(* IEC 61131-3 sources: -3/Library, 1 file *)

(* ---- Library.fun ---- *)
FUNCTION_BLOCK FB_Motor (*TODO: Add your comment here*) (*$GROUP=User,$CAT=User,$GROUPICON=User.png,$CATICON=User.png*)
	VAR_INPUT
		in : REAL;
	END_VAR
	VAR_OUTPUT
		out_w : REAL;
		out_phi : REAL;
	END_VAR
	VAR
		k_e : REAL;
		T_m : REAL;
		dt : REAL;
		integrator : FB_Integrator;
		integrator_phi : FB_Integrator;
	END_VAR
END_FUNCTION_BLOCK

FUNCTION_BLOCK FB_Integrator (*TODO: Add your comment here*) (*$GROUP=User,$CAT=User,$GROUPICON=User.png,$CATICON=User.png*)
	VAR_INPUT
		in : REAL;
		dt : REAL;
	END_VAR
	VAR_OUTPUT
		out : REAL;
	END_VAR
	VAR
		state : REAL := 0.0;
	END_VAR
END_FUNCTION_BLOCK

FUNCTION_BLOCK FB_Controller (* *) (*$GROUP=User,$CAT=User,$GROUPICON=User.png,$CATICON=User.png*)
	VAR_INPUT
		in : REAL;
	END_VAR
	VAR_OUTPUT
		out : REAL;
	END_VAR
	VAR
		k_i : REAL;
		sum : REAL;
		k_p : REAL;
		dt : REAL;
		max_abs_value : REAL;
		integrator : FB_Integrator;
		last_sum : REAL;
	END_VAR
END_FUNCTION_BLOCK

FUNCTION_BLOCK FB_Endswitch (*TODO: Add your comment here*) (*$GROUP=User,$CAT=User,$GROUPICON=User.png,$CATICON=User.png*)
	VAR_INPUT
		in : REAL;
		neg_value : REAL;
		pos_value : REAL;
	END_VAR
	VAR_OUTPUT
		neg_reached : BOOL;
		pos_reached : BOOL;
	END_VAR
END_FUNCTION_BLOCK

FUNCTION_BLOCK FB_Axis (*TODO: Add your comment here*) (*$GROUP=User,$CAT=User,$GROUPICON=User.png,$CATICON=User.png*)
	VAR_INPUT
		u : REAL;
		reset_error : BOOL;
		endswitch_a_reached : BOOL;
		endswitch_b_reached : BOOL;
		pwm_percentage : SINT;
	END_VAR
	VAR_OUTPUT
		reset_counter : BOOL;
		pwm_value : INT;
	END_VAR
	VAR_OUTPUT RETAIN
		counter : INT;
	END_VAR
	VAR_OUTPUT
		speed : REAL;
	END_VAR
	VAR
		i : INT;
		last_counter : INT;
		dir : BOOL;
		spid : REAL;
		k : INT;
	END_VAR
END_FUNCTION_BLOCK

{REDUND_ERROR} FUNCTION_BLOCK FB_Regulator (*TODO: Add your comment here*) (*$GROUP=User,$CAT=User,$GROUPICON=User.png,$CATICON=User.png*)
	VAR_INPUT
		e : REAL;
	END_VAR
	VAR_OUTPUT
		u : REAL;
	END_VAR
	VAR
		k_p : REAL;
		k_i : REAL;
		integrator : FB_Integrator;
		iyOld : REAL;
		max_abc_value : REAL := 24;
		dt : REAL;
		x : REAL;
	END_VAR
END_FUNCTION_BLOCK

{REDUND_ERROR} FUNCTION_BLOCK Pos (*TODO: Add your comment here*) (*$GROUP=User,$CAT=User,$GROUPICON=User.png,$CATICON=User.png*)
	VAR_INPUT
		enable : BOOL;
	END_VAR
END_FUNCTION_BLOCK
